Fanuc KAREL source: RIF_COMMANDS.KL

PROGRAM RIF_COMMANDS
%STACKSIZE = 4000
%NOLOCKGROUP
%NOPAUSE=ERROR+COMMAND+TPENABLE
%ENVIRONMENT uif
%ENVIRONMENT sysdef
%ENVIRONMENT memo
%ENVIRONMENT kclop
%ENVIRONMENT bynam
%ENVIRONMENT fdev
%ENVIRONMENT flbt
%ENVIRONMENT regope
-- %INCLUDE klevccdf
-- %INCLUDE klevkeys
-- %INCLUDE klevkmsk
CONST
    cc_home = 137
    cc_clear_win = 128

    RIF_RANGE = 25
    NORM_RIFTEK = 16384

    RIFTEK_DEFAULT_COMMAND = 128
VAR
    data_type   : INTEGER
    int_value : INTEGER
    real_value : REAL
    str_value : STRING[20]
    status : INTEGER

	INDEX : INTEGER
    comm_file : FILE

    ----INPUT PARAMETERS----
    COMMAND_TYPE : INTEGER

    PARAMETER_SIZE_IN_BYTES : INTEGER
    PARAMETER_FIRST_BYTE_CODE : INTEGER
    PARAMETER_VALUE : INTEGER
    PARAMETERS_FIRST_REGISTER : INTEGER
    ----INPUT PARAMETERS----



    REQUEST_SIZE : INTEGER
    REQUEST_PARAMETER_ARR_TAKE_INDEX : INTEGER
    REQUEST_PARAMETER_ARR_TAKE_LENGTH : INTEGER
    REQUSET_PARAMETER_CODE_ARRAY : ARRAY[20] OF BYTE
    REQUSET_PARAMETER_VALUE_ARRAY : ARRAY[20] OF BYTE
    REQUEST_ARRAY : ARRAY[20] OF BYTE
    REQUEST_ARRAY_PUSH_INDEX : INTEGER

    RESPONSE_SIZE : INTEGER
    RESPONSE_ARRAY : ARRAY[20] OF BYTE
    RESPONSE_PARAMETER_VALUE_ARRAY : ARRAY[20] OF BYTE
    RESPONSE_PARAMETER_ARR_PUSH_INDEX : INTEGER


    --DEVICE INFO--
	--TYPE
	--RANGE_INFO = STRUCTURE
	DEVICE_TYPE : REAL
	PO_VERSION : REAL
    SERIAL_NUMBER : REAL
    BASE_DISTANCE : REAL
    RANGE : REAL
    --ENDSTRUCTURE
    --DEVICE INFO--

    DISTANCE : REAL


    ----POST ERRORS----
    ROUTINE POSTERR(cause : STRING; status : INTEGER) &
    FROM CUST_ERRORS
    ROUTINE POST_CUST_ERR(cause : STRING) &
    FROM CUST_ERRORS
    ----POST ERRORS----

    ----READ INTEGER PARAMETER----
    ROUTINE GET_TPE_INT_PARAMETER(number : INTEGER) : INTEGER &
    FROM CUST_READ_PARAMS
    ----READ INTEGER PARAMETER----

    ----PARAMS CONVERTS----
    ROUTINE CNV_DECIMAL_PARAM_TO_BYTE_ARRAY(param : INTEGER; param_size : INTEGER) : ARRAY OF BYTE &
    FROM CONVERT_PARAMS

    ROUTINE CNV_DECIMAL_PARAM_CODE_TO_BYTE_ARRAY(param_code : INTEGER; param_size : INTEGER) : ARRAY OF BYTE &
    FROM CONVERT_PARAMS

    ROUTINE READ_PARAMETER_FROM_BYTE_ARRAY(response : ARRAY OF BYTE; start_byte_number : INTEGER; bytes_count : INTEGER) : INTEGER &
    FROM CONVERT_PARAMS

    ----PARAMS CONVERTS----

    ROUTINE CLEAR_ARR_TO_END(arr : ARRAY OF BYTE; START_INDEX : INTEGER) &
    FROM CUST_ARR_UTIL

    ROUTINE PUSH_TO_ARRAY(dest_arr : ARRAY OF BYTE; dest_arr_insert_index : INTEGER; source_arr : ARRAY OF BYTE; source_arr_take_index : INTEGER; source_arr_take_length : INTEGER) &
    FROM CUST_ARR_UTIL


-------------------------------------------------------------------------------------------------------
---------------------------------------RIFTEK MESSAGES UTIL ROUTINES-----------------------------------
--WRITE COMMAND CODE AND NETWORK ADDRESS TO REQUEST ARRAY
ROUTINE WRITE_COMMAND_TO_REQUEST_ARRAY(arr : ARRAY OF BYTE; c_type : INTEGER)
BEGIN
    arr[1] = 1
    arr[2] = RIFTEK_DEFAULT_COMMAND + c_type
END WRITE_COMMAND_TO_REQUEST_ARRAY
--SEND REQUEST TO SPECIFIED PORT(FILE) WITH REQEST ARRAY DATA
ROUTINE SEND_REQUEST(req_bytes : ARRAY OF BYTE;  req_size : INTEGER; c_file : FILE)
VAR
    index : INTEGER
BEGIN
    FOR INDEX = 1 TO req_size DO
        --WRITE ('RQ ',req_bytes[INDEX]::1,CR)
        WRITE c_file(req_bytes[INDEX]::1)
    ENDFOR

    STATUS = IO_STATUS(comm_file)
    WRITE('FILE STATUS  =  ',STATUS,CR)

END SEND_REQUEST
--READ RESPONCE FROM SPECIFIED PORT(FILE) AND WRITE RESPONSE DATA TO RESPONSE ARRRAY
ROUTINE READ_RESPONSE(res_bytes : ARRAY OF BYTE; res_size : INTEGER; c_file : FILE)
VAR
    IND : INTEGER
BEGIN
    FOR IND = 1 TO res_size DO
        READ c_file(res_bytes[IND]::1)
        --WRITE('RS', res_bytes[IND]::1, CR)
    ENDFOR

    STATUS = IO_STATUS(comm_file)
    WRITE('FILE STATUS  =  ', STATUS, CR)

END READ_RESPONSE
---------------------------------------RIFTEK MESSAGES UTIL ROUTINES-----------------------------------
-------------------------------------------------------------------------------------------------------

----DEVICE IDENTIFICATION ROUTINE----
ROUTINE DEVICE_IDENTIFICATION(c_file : FILE; register : INTEGER)
BEGIN
    -- GET REGISTER
    PARAMETERS_FIRST_REGISTER = register

    COMMAND_TYPE = 1
    REQUEST_SIZE = 2
    RESPONSE_SIZE = 16
    WRITE_COMMAND_TO_REQUEST_ARRAY(REQUEST_ARRAY, COMMAND_TYPE)
    FOR INDEX = 1 TO REQUEST_SIZE DO
        WRITE(REQUEST_ARRAY[INDEX],CR)
    ENDFOR
    SEND_REQUEST(REQUEST_ARRAY, REQUEST_SIZE, c_file)
    READ_RESPONSE(RESPONSE_ARRAY, RESPONSE_SIZE, c_file)

    --DEVICE TYPE--
    DEVICE_TYPE =  READ_PARAMETER_FROM_BYTE_ARRAY(RESPONSE_ARRAY, 1, 1)
    SET_REAL_REG(PARAMETERS_FIRST_REGISTER, DEVICE_TYPE, STATUS)

    --PO VERSION--
    PO_VERSION = READ_PARAMETER_FROM_BYTE_ARRAY(RESPONSE_ARRAY, 3, 1)
    SET_REAL_REG(PARAMETERS_FIRST_REGISTER + 1, PO_VERSION, STATUS)

    --SERIAL NUMBER--
    SERIAL_NUMBER = READ_PARAMETER_FROM_BYTE_ARRAY(RESPONSE_ARRAY, 5, 2)
    SET_REAL_REG(PARAMETERS_FIRST_REGISTER + 2, SERIAL_NUMBER, STATUS)

    --BASE DISTANCE--
    BASE_DISTANCE = READ_PARAMETER_FROM_BYTE_ARRAY(RESPONSE_ARRAY, 9, 2)
    SET_REAL_REG(PARAMETERS_FIRST_REGISTER + 3, BASE_DISTANCE, STATUS)

    --RANGE--
    RANGE = READ_PARAMETER_FROM_BYTE_ARRAY(RESPONSE_ARRAY, 13, 2)
    SET_REAL_REG(PARAMETERS_FIRST_REGISTER + 4, RANGE, STATUS)
END DEVICE_IDENTIFICATION
----READ PARAMETER ROUTINE----
ROUTINE READ_PARAMETER_VALUE(c_file : FILE; size : INTEGER; code : INTEGER; register : INTEGER)
VAR
    IN_INDEX : INTEGER
BEGIN
    --READ PARAMETER SIZE (BYTES)
    PARAMETER_SIZE_IN_BYTES = size

    --READ PARAMETER FIRST BYTE CODE INT OR STRING
    PARAMETER_FIRST_BYTE_CODE = code

    --READ REGISTER
    PARAMETERS_FIRST_REGISTER = register

    COMMAND_TYPE = 2
    REQUEST_SIZE = 4
    RESPONSE_SIZE = 2

    WRITE_COMMAND_TO_REQUEST_ARRAY(REQUEST_ARRAY, COMMAND_TYPE)

    REQUSET_PARAMETER_CODE_ARRAY = CNV_DECIMAL_PARAM_CODE_TO_BYTE_ARRAY(PARAMETER_FIRST_BYTE_CODE, PARAMETER_SIZE_IN_BYTES)

    -- FOR INDEX = 1 TO PARAMETER_SIZE_IN_BYTES * 4 DO
    --     WRITE(REQUSET_PARAMETER_CODE_ARRAY[INDEX], ' ')
    -- ENDFOR
    -- WRITE(CR)

    REQUEST_ARRAY_PUSH_INDEX = 3
    REQUEST_PARAMETER_ARR_TAKE_INDEX = 1
    REQUEST_PARAMETER_ARR_TAKE_LENGTH = 2
    RESPONSE_PARAMETER_ARR_PUSH_INDEX = 1

    FOR INDEX = 1 TO PARAMETER_SIZE_IN_BYTES DO
        PUSH_TO_ARRAY(REQUEST_ARRAY, REQUEST_ARRAY_PUSH_INDEX, REQUSET_PARAMETER_CODE_ARRAY, REQUEST_PARAMETER_ARR_TAKE_INDEX, REQUEST_PARAMETER_ARR_TAKE_LENGTH)
        SEND_REQUEST(REQUEST_ARRAY, REQUEST_SIZE, c_file)

        READ_RESPONSE(RESPONSE_ARRAY, RESPONSE_SIZE, c_file)

        PUSH_TO_ARRAY(RESPONSE_PARAMETER_VALUE_ARRAY, RESPONSE_PARAMETER_ARR_PUSH_INDEX, RESPONSE_ARRAY, 1, RESPONSE_SIZE)

        REQUEST_PARAMETER_ARR_TAKE_INDEX = REQUEST_PARAMETER_ARR_TAKE_INDEX + 2
        RESPONSE_PARAMETER_ARR_PUSH_INDEX = RESPONSE_PARAMETER_ARR_PUSH_INDEX + 2
    ENDFOR

    FOR INDEX = 1 TO PARAMETER_SIZE_IN_BYTES * 2 DO
        WRITE(RESPONSE_PARAMETER_VALUE_ARRAY[INDEX], ' ')
    ENDFOR


    PARAMETER_VALUE = READ_PARAMETER_FROM_BYTE_ARRAY(RESPONSE_PARAMETER_VALUE_ARRAY, 1, PARAMETER_SIZE_IN_BYTES)

    SET_INT_REG(PARAMETERS_FIRST_REGISTER, PARAMETER_VALUE, STATUS)

    CLEAR_ARR_TO_END(REQUSET_PARAMETER_CODE_ARRAY, 1)
    CLEAR_ARR_TO_END(REQUEST_ARRAY, 1)
    CLEAR_ARR_TO_END(RESPONSE_ARRAY, 1)
    CLEAR_ARR_TO_END(RESPONSE_PARAMETER_VALUE_ARRAY, 1)
END READ_PARAMETER_VALUE
----WRITE PARAMETER ROUTINE----
ROUTINE WRITE_PARAMETER_VALUE(c_file : FILE; size : INTEGER; code : INTEGER; value : INTEGER)
VAR
    IN_INDEX : INTEGER
BEGIN
    --READ PARAMETER SIZE (BYTES)
    PARAMETER_SIZE_IN_BYTES = size

    --READ PARAMETER FIRST BYTE CODE INT OR STRING
    PARAMETER_FIRST_BYTE_CODE = code

    --READ PARAMETER VALUE
    PARAMETER_VALUE = value
    COMMAND_TYPE = 3
    REQUEST_SIZE = 6

    --WRITE REQUEST CODE TO REQUEST ARRAY
    WRITE_COMMAND_TO_REQUEST_ARRAY(REQUEST_ARRAY, COMMAND_TYPE)
    --WTITE PARAMETER CODE TO PARAMETER ARRAY
    REQUSET_PARAMETER_CODE_ARRAY = CNV_DECIMAL_PARAM_CODE_TO_BYTE_ARRAY(PARAMETER_FIRST_BYTE_CODE, PARAMETER_SIZE_IN_BYTES)

    -- FOR IN_INDEX = 1 TO PARAMETER_SIZE_IN_BYTES * 2 DO
    --     WRITE(REQUSET_PARAMETER_CODE_ARRAY[IN_INDEX], ' ')
    -- ENDFOR
    -- WRITE(CR)

    --WTITE PARAMETER VALUE TO PARAMETER ARRAY
    REQUSET_PARAMETER_VALUE_ARRAY = CNV_DECIMAL_PARAM_TO_BYTE_ARRAY(PARAMETER_VALUE, PARAMETER_SIZE_IN_BYTES)

    -- FOR IN_INDEX = 1 TO PARAMETER_SIZE_IN_BYTES * 2 DO
    --     WRITE(REQUSET_PARAMETER_VALUE_ARRAY[IN_INDEX], ' ')
    -- ENDFOR
    -- WRITE(CR)

    REQUEST_ARRAY_PUSH_INDEX = 3
    REQUEST_PARAMETER_ARR_TAKE_INDEX = PARAMETER_SIZE_IN_BYTES * 2 - 1
    REQUEST_PARAMETER_ARR_TAKE_LENGTH = 2

    FOR INDEX = 1 TO PARAMETER_SIZE_IN_BYTES DO
        PUSH_TO_ARRAY(REQUEST_ARRAY, REQUEST_ARRAY_PUSH_INDEX, REQUSET_PARAMETER_CODE_ARRAY, REQUEST_PARAMETER_ARR_TAKE_INDEX, REQUEST_PARAMETER_ARR_TAKE_LENGTH)
        PUSH_TO_ARRAY(REQUEST_ARRAY, REQUEST_ARRAY_PUSH_INDEX + 2, REQUSET_PARAMETER_VALUE_ARRAY, REQUEST_PARAMETER_ARR_TAKE_INDEX, REQUEST_PARAMETER_ARR_TAKE_LENGTH)
        FOR IN_INDEX = 1 TO REQUEST_SIZE DO
            WRITE(REQUEST_ARRAY[IN_INDEX], ' ')
        ENDFOR
        WRITE(CR)
        SEND_REQUEST(REQUEST_ARRAY, REQUEST_SIZE, c_file)

        REQUEST_PARAMETER_ARR_TAKE_INDEX = REQUEST_PARAMETER_ARR_TAKE_INDEX - 2
    ENDFOR

    CLEAR_ARR_TO_END(REQUSET_PARAMETER_CODE_ARRAY, 1)
    CLEAR_ARR_TO_END(REQUSET_PARAMETER_VALUE_ARRAY, 1)
    CLEAR_ARR_TO_END(REQUEST_ARRAY, 1)
END WRITE_PARAMETER_VALUE
----SAVE FLASH MEMORY----
ROUTINE SAVE_FLASH_MEMORY(c_file :FILE; register : INTEGER)
BEGIN
    PARAMETERS_FIRST_REGISTER = register
    PARAMETER_FIRST_BYTE_CODE = 170
    COMMAND_TYPE = 4
    REQUEST_SIZE = 4
    RESPONSE_SIZE = 2

    WRITE_COMMAND_TO_REQUEST_ARRAY(REQUEST_ARRAY, COMMAND_TYPE)
    REQUSET_PARAMETER_CODE_ARRAY = CNV_DECIMAL_PARAM_CODE_TO_BYTE_ARRAY(PARAMETER_FIRST_BYTE_CODE, 1)

    REQUEST_ARRAY_PUSH_INDEX = 3
    REQUEST_PARAMETER_ARR_TAKE_INDEX = 1
    REQUEST_PARAMETER_ARR_TAKE_LENGTH = 2
    RESPONSE_PARAMETER_ARR_PUSH_INDEX = 1

    PUSH_TO_ARRAY(REQUEST_ARRAY, REQUEST_ARRAY_PUSH_INDEX, REQUSET_PARAMETER_CODE_ARRAY, REQUEST_PARAMETER_ARR_TAKE_INDEX, REQUEST_PARAMETER_ARR_TAKE_LENGTH)
    SEND_REQUEST(REQUEST_ARRAY, REQUEST_SIZE, c_file)
    READ_RESPONSE(RESPONSE_ARRAY, RESPONSE_SIZE, c_file)

    PARAMETER_VALUE = READ_PARAMETER_FROM_BYTE_ARRAY(RESPONSE_ARRAY, 1, PARAMETER_SIZE_IN_BYTES)
    SET_INT_REG(PARAMETERS_FIRST_REGISTER, PARAMETER_VALUE, STATUS)

    CLEAR_ARR_TO_END(REQUSET_PARAMETER_CODE_ARRAY, 1)
    CLEAR_ARR_TO_END(REQUEST_ARRAY, 1)
    CLEAR_ARR_TO_END(RESPONSE_ARRAY, 1)
END SAVE_FLASH_MEMORY
----LOAD DEFAULT PARAMETERS  IN FLASH MEMORY----
ROUTINE LOAD_DEFAULT_PARAMETERS(c_file :FILE; register : INTEGER)
BEGIN
    PARAMETERS_FIRST_REGISTER = register
    PARAMETER_FIRST_BYTE_CODE = 105
    COMMAND_TYPE = 4
    REQUEST_SIZE = 4
    RESPONSE_SIZE = 2

    WRITE_COMMAND_TO_REQUEST_ARRAY(REQUEST_ARRAY, COMMAND_TYPE)
    REQUSET_PARAMETER_CODE_ARRAY = CNV_DECIMAL_PARAM_CODE_TO_BYTE_ARRAY(PARAMETER_FIRST_BYTE_CODE, 1)

    REQUEST_ARRAY_PUSH_INDEX = 3
    REQUEST_PARAMETER_ARR_TAKE_INDEX = 1
    REQUEST_PARAMETER_ARR_TAKE_LENGTH = 2
    RESPONSE_PARAMETER_ARR_PUSH_INDEX = 1

    PUSH_TO_ARRAY(REQUEST_ARRAY, REQUEST_ARRAY_PUSH_INDEX, REQUSET_PARAMETER_CODE_ARRAY, REQUEST_PARAMETER_ARR_TAKE_INDEX, REQUEST_PARAMETER_ARR_TAKE_LENGTH)
    SEND_REQUEST(REQUEST_ARRAY, REQUEST_SIZE, c_file)
    READ_RESPONSE(RESPONSE_ARRAY, RESPONSE_SIZE, c_file)

    PARAMETER_VALUE = READ_PARAMETER_FROM_BYTE_ARRAY(RESPONSE_ARRAY, 1, PARAMETER_SIZE_IN_BYTES)
    SET_INT_REG(PARAMETERS_FIRST_REGISTER, PARAMETER_VALUE, STATUS)

    CLEAR_ARR_TO_END(REQUSET_PARAMETER_CODE_ARRAY, 1)
    CLEAR_ARR_TO_END(REQUEST_ARRAY, 1)
    CLEAR_ARR_TO_END(RESPONSE_ARRAY, 1)
END LOAD_DEFAULT_PARAMETERS
----RESULT SNAPPING----
ROUTINE RESULT_SNAPPING(c_file : FILE)
BEGIN
    COMMAND_TYPE = 5
    REQUEST_SIZE = 2

    WRITE_COMMAND_TO_REQUEST_ARRAY(REQUEST_ARRAY, COMMAND_TYPE)
    SEND_REQUEST(REQUEST_ARRAY, REQUEST_SIZE, c_file)
END RESULT_SNAPPING
----GET RANGE VALUE----
ROUTINE GET_RANGE(c_file : FILE; register : INTEGER)
BEGIN
    --GET REGISTER
    PARAMETERS_FIRST_REGISTER = register
    COMMAND_TYPE = 6
    REQUEST_SIZE = 2
    RESPONSE_SIZE = 4

    WRITE_COMMAND_TO_REQUEST_ARRAY(REQUEST_ARRAY, COMMAND_TYPE)
    SEND_REQUEST(REQUEST_ARRAY, REQUEST_SIZE, c_file)
    READ_RESPONSE(RESPONSE_ARRAY, RESPONSE_SIZE, c_file)

    DISTANCE = READ_PARAMETER_FROM_BYTE_ARRAY(RESPONSE_ARRAY, 1, RESPONSE_SIZE)
    DISTANCE = DISTANCE * RIF_RANGE / NORM_RIFTEK

    SET_REAL_REG(PARAMETERS_FIRST_REGISTER, DISTANCE, STATUS)
END GET_RANGE
----START RANGE THREAD----
ROUTINE START_RANGE_THREAD(c_file : FILE)
VAR
    STOP_SIGNAL : BOOLEAN
BEGIN
    COMMAND_TYPE = 7
    REQUEST_SIZE = 2
    RESPONSE_SIZE = 4
    WRITE_COMMAND_TO_REQUEST_ARRAY(REQUEST_ARRAY, COMMAND_TYPE)
    SEND_REQUEST(REQUEST_ARRAY, REQUEST_SIZE, c_file)
END START_RANGE_THREAD
----READ VALUE FROM RANGE THREAD----
ROUTINE READ_RANGE_THREAD(c_file : FILE; register : INTEGER) : REAL
BEGIN
    --GET REGISTER
    PARAMETERS_FIRST_REGISTER = register
    REQUEST_SIZE = 2
    RESPONSE_SIZE = 4
    READ_RESPONSE(RESPONSE_ARRAY, RESPONSE_SIZE, c_file)

    DISTANCE = READ_PARAMETER_FROM_BYTE_ARRAY(RESPONSE_ARRAY, 1, RESPONSE_SIZE)
    DISTANCE = DISTANCE * RIF_RANGE / NORM_RIFTEK

    SET_REAL_REG(PARAMETERS_FIRST_REGISTER, DISTANCE, STATUS)
    RETURN (DISTANCE)
END READ_RANGE_THREAD
----STOP RANGE THREAD----
ROUTINE STOP_RANGE_THREAD(c_file: FILE)
BEGIN
    COMMAND_TYPE = 8
    REQUEST_SIZE = 2

    WRITE_COMMAND_TO_REQUEST_ARRAY(REQUEST_ARRAY, COMMAND_TYPE)
    SEND_REQUEST(REQUEST_ARRAY, REQUEST_SIZE, c_file)
END STOP_RANGE_THREAD
-------------------------------------RIFTEK QUERY CODES ROUTINES---------------------------------------
-------------------------------------------------------------------------------------------------------
BEGIN
END RIF_COMMANDS
